FUNCTION_BLOCK TickGen
  (* Standard: 61499-2 *)
  (* Version 0.1, 2017-00-29, hpea485, UOA *)
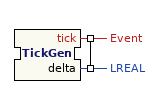
  EVENT_OUTPUT
    tick WITH delta;
  END_EVENT
  VAR_OUTPUT
    delta : LREAL;
  END_VAR
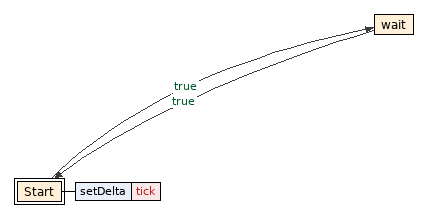
  EC_STATES
    Start : setDelta -> tick;
    wait;
  END_STATES
  EC_TRANSITIONS
    Start TO wait := true;
    wait TO Start := true;
  END_TRANSITIONS
  ALGORITHM setDelta IN C:
me->delta = 0.10;
  END_ALGORITHM
END_FUNCTION_BLOCK
